// TIA Portal V20 export
// export: Created 2025-12-01T14:56:21.5930778Z, ExportSetting None, DisplayName Totally Integrated Automation Portal, DisplayVersion V20 Update 3, DisplayName TIA Portal Openness, DisplayVersion V20 Update 3, DisplayName TIA Portal Version Control Interface, DisplayVersion V20 Update 3, DisplayName STEP 7 Professional, DisplayVersion V20 Update 3, DisplayName STEP 7 Safety, DisplayVersion V20 Update 2, DisplayName WinCC Basic/Comfort/Advanced, DisplayVersion V20 Update 3, DisplayName WinCC Professional, DisplayVersion V20 Update 3, DisplayName WinCC Unified, DisplayVersion V20 Update 3
TYPE "EstadoMaquina_DesPaletizadoManual"
   STRUCT
      Etapa_Reset : Bool;   // Etapa MAQUINA en RESET
      Etapa_EnReposo : Bool;   // Etapa MAQUINA en REPOSO
      Etapa_EnMovimiento : Bool;   // Etapa MAQUINA en MOVIMIENTO
      Etapa_libre_03 : Bool;   // ...
      Etapa_libre_04 : Bool;   // ...
      Etapa_libre_05 : Bool;   // ...
      Etapa_libre_06 : Bool;   // ...
      Etapa_libre_07 : Bool;   // ...
      PaletaEnPuesto : Bool;   // ...
      Puesto_NuevaCapa : Bool;   // ...
      Puesto_MovManual : Bool;   // ...
      Elev_MovCarga : Bool;   // ...
      Elev_MovDesCarga : Bool;   // ...
      Elev_MovEnPuesto : Bool;   // ...
      Etapa_libre_14 : Bool;   // ...
      Manual : Bool;   // MAQUINA EN MANUAL
      Err_TermicoElevacion : Bool;   // 01. ERROR
      Byte2_bit1 : Bool;   // 02. ERROR
      Byte2_bit2 : Bool;   // 03. ERROR
      Err_PosicionCargaDesCarga : Bool;   // 04. ERROR
      Err_ReferenciaOK : Bool;   // 05. ERROR
      Err_TimeOutElevacion : Bool;   // 06. ERROR
      Byte2_bit6 : Bool;   // 07. ERROR
      Byte2_bit7 : Bool;   // 08. ERROR
      Byte3_bit0 : Bool;   // 09. ERROR
      Byte3_bit1 : Bool;   // 10. ERROR
      Byte3_bit2 : Bool;   // 11. ERROR
      Byte3_bit3 : Bool;   // 12. ERROR
      Byte3_bit4 : Bool;   // 13. ERROR
      Byte3_bit5 : Bool;   // 14. ERROR
      Byte3_bit6 : Bool;   // 15. ERROR
      Byte3_bit7 : Bool;   // 16. ERROR
      Err_SeguridadArriba : Bool;   // 17. ERROR
      Err_SeguridadAbajo : Bool;   // 18. ERROR
      Err_RoturaDeCadena : Bool;   // 19. ERROR
      Byte4_bit3 : Bool;   // 20. ERROR
      Err_Protrusion : Bool;   // 21. ERROR
      Byte4_bit5 : Bool;   // 22. ERROR
      Byte4_bit6 : Bool;   // 23. ERROR
      Byte4_bit7 : Bool;   // 24. ERROR
      Byte5_bit0 : Bool;   // 25. ERROR
      Byte5_bit1 : Bool;   // 26. ERROR
      Byte5_bit2 : Bool;   // 27. ERROR
      Byte5_bit3 : Bool;   // 28. ERROR
      Byte5_bit4 : Bool;   // 29. ERROR
      Byte5_bit5 : Bool;   // 30. ERROR
      Byte5_bit6 : Bool;   // 31. ERROR
      Byte5_bit7 : Bool;   // 32. ERROR
      Byte6_bit0 : Bool;   // 33. ERROR
      Byte6_bit1 : Bool;   // 34. ERROR
      Byte6_bit2 : Bool;   // 35. ERROR
      Byte6_bit3 : Bool;   // 36. ERROR
      Byte6_bit4 : Bool;   // 37. ERROR
      Byte6_bit5 : Bool;   // 38. ERROR
      Byte6_bit6 : Bool;   // 39. ERROR
      Error_MAQx : Bool;   // Marca General Errol
      TermicoFreno : Bool;   // Entrada 1
      Byte7_bit1 : Bool;   // Entrada 2
      Byte7_bit2 : Bool;   // Entrada 3
      Byte7_bit3 : Bool;   // Entrada 4
      Byte7_bit4 : Bool;   // Entrada 5
      Byte7_bit5 : Bool;   // Entrada 6
      Byte7_bit6 : Bool;   // Entrada 7
      Byte7_bit7 : Bool;   // Entrada 8
      Byte8_bit0 : Bool;   // Entrada 9
      Byte8_bit1 : Bool;   // Entrada 10
      Byte8_bit2 : Bool;   // Entrada 11
      Byte8_bit3 : Bool;   // Entrada 12
      Byte8_bit4 : Bool;   // Entrada 13
      Byte8_bit5 : Bool;   // Entrada 14
      Byte8_bit6 : Bool;   // Entrada 15
      Byte8_bit7 : Bool;   // Entrada 16
      Protrusion : Bool;   // Entrada 17
      SeguridadArriba : Bool;   // Entrada 18
      SeguridadAbajo : Bool;   // Entrada 19
      Byte9_bit3 : Bool;   // Entrada 20
      Elev_ReferenciaOK : Bool;   // Entrada 21
      Byte9_bit5 : Bool;   // Entrada 22
      Byte9_bit6 : Bool;   // Entrada 23
      Byte9_bit7 : Bool;   // Entrada 24
      Elev_Subiendo : Bool;   // Salida 1
      Elev_Bajando : Bool;   // Salida 2
      Byte10_bit2 : Bool;   // Salida 3
      Byte10_bit3 : Bool;   // Salida 4
      Byte10_bit4 : Bool;   // Salida 5
      Byte10_bit5 : Bool;   // Salida 6
      Byte10_bit6 : Bool;   // Salida 7
      Byte10_bit7 : Bool;   // Salida 8
      Byte11_bit0 : Bool;   // Salida 9
      Byte11_bit1 : Bool;   // Salida 10
      Byte11_bit2 : Bool;   // Salida 11
      Byte11_bit3 : Bool;   // Salida 12
      Byte11_bit4 : Bool;   // Salida 13
      Byte11_bit5 : Bool;   // Salida 14
      Byte11_bit6 : Bool;   // Salida 15
      Byte11_bit7 : Bool;   // Salida 16
      Byte12_bit0 : Bool;   // Salida 17
      Byte12_bit1 : Bool;   // Salida 18
      Fin_VI : Bool;   // Fin de Vehiculo
      Paro_Blando : Bool;   // Maquina en paro blando
      Byte12_bit4 : Bool;   // ...
      Byte12_bit5 : Bool;   // ...
      Byte12_bit6 : Bool;   // ...
      Byte12_bit7 : Bool;   // ...
      Pulsador_Subir : Bool;   // ...
      Pulsador_Bajar : Bool;   // ...
      Pulsador_NuevaCapa : Bool;   // ...
      Barrera_Arriba : Bool;   // ...
      pHs_PisoCarga : Bool;   // ...
      pHs_PisoDesCarga : Bool;   // ...
      Byte13_bit6 : Bool;   // ...
      Baliza : Bool;   // ...
      pHsGalibo_01 : Bool;   // ...
      pHsGalibo_02 : Bool;   // ...
      pHsGalibo_03 : Bool;   // ...
      pHsGalibo_04 : Bool;   // ...
      pHsAlturaCota : Bool;   // ...
      pHsAnchura : Bool;   // ...
      pHsAlturaMax_01 : Bool;   // ...
      pHsAlturaMax_02 : Bool;   // ...
      RoturaCadena_01 : Bool;   // ...
      RoturaCadena_02 : Bool;   // ...
      RoturaCadena_03 : Bool;   // ...
      RoturaCadena_04 : Bool;   // ...
      Byte15_bit4 : Bool;   // ...
      Byte15_bit5 : Bool;   // ...
      Byte15_bit6 : Bool;   // ...
      Byte15_bit7 : Bool;   // ...
   END_STRUCT;
END_TYPE
